(* CoDeSys 2.3.9.37 project: CapB_5.pro *)
(* Libraries: Standard.lib 4.10.05 12:14:46, IecSfc.lib 13.4.06 16:51:28, SYSLIBCALLBACK.LIB 26.9.08 17:43:52 *)

(* Task configuration *)
TASK NewTask (PRIORITY := 1, INTERVAL := T#100ms);
	PLC_PRG
END_TASK

(* POU PLC_PRG, ST *)
PROGRAM PLC_PRG
VAR
   Nivel: REAL:=2.0;
   ValvulaEntrada:BOOL;
   ValvulaSalida:BOOL;
   CaudalEntrada:REAL:=0;
   CaudalSalida:REAL:=0;
   Area:REAL:=1;
   IntT:REAL:=0.1;
   KEntrada:REAL:=0.1;
   KSalida:REAL:=0.2;
	Neto: REAL;
	Nivellnf:REAL:=0;
	NivelSup:REAL:=5;
END_VAR
CaudalEntrada:=BOOL_TO_INT(ValvulaEntrada)*KEntrada;
CaudalSalida:=BOOL_TO_INT(ValvulaSalida)*KSalida;
Neto:=(CaudalEntrada-CaudalSalida);
IF (Neto<0AND Nivel>Nivellnf) OR (Neto>0 AND Nivel<NivelSup) THEN
   Nivel:=Nivel+IntT*Neto;
END_IF
END_PROGRAM

(* Visualisation Deposito
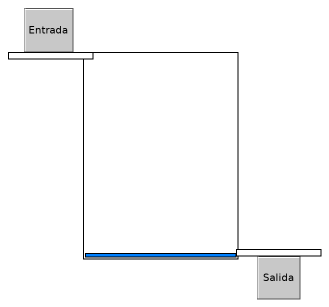
button at (20,69)-(69,113): text "Entrada"; toggles PLC_PRG.ValvulaEntrada
button at (253,317)-(296,360): text "Salida"; toggles PLC_PRG.ValvulaSalida
rectangle at (81,314)-(232,318): top -40*PLC_PRG.Nivel
rectangle at (232,310)-(317,317): alarm colour if PLC_PRG.ValvulaSalida AND PLC_PRG.Nivel>0
rectangle at (4,113)-(89,120): alarm colour if PLC_PRG.ValvulaEntrada
1 more shapes without text or variables
1 elements of other kinds (tables, trends, ...) not read
*)
